Omron CX-Programmer project NewProject (CX-Programmer 9.75)

# PLC NewPLC1: CP1E E20

## Program NewProgram1 (cyclic task 0)

### Section Section1

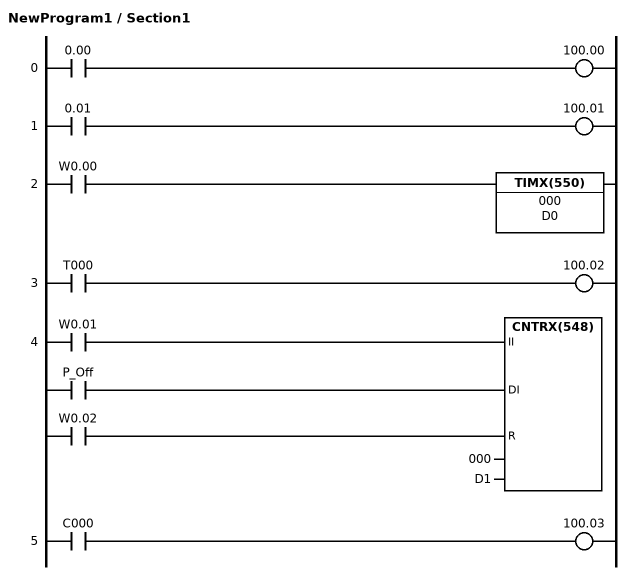
; rung 0
LD 0.00
OUT 100.00
; rung 1
LD 0.01
OUT 100.01
; rung 2
LD W0.00
TIMX(550) 000 D0
; rung 3
LD T000
OUT 100.02
; rung 4
LD W0.01
LD P_Off
LD W0.02
CNTRX(548) 000 D1
; rung 5
LD C000
OUT 100.03

### Section END
; rung 0
END(001)